SUBAPPLICATION GreenWhiteBackground_Seitenschieber (* Subapplication Type *)
  (* Standard: 61499-2 *)
  (* Version 1.0, 2023-02-06, franz *)
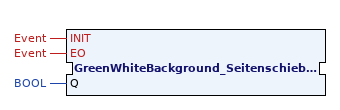
  EVENT_INPUT
    INIT;
    EO;
  END_EVENT
  VAR_INPUT
    Q : BOOL;
  END_VAR
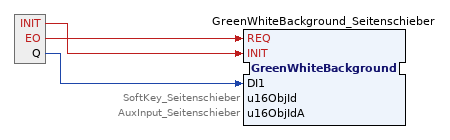
  SUBAPPS
    GreenWhiteBackground_Seitenschieber : GreenWhiteBackground(u16ObjId := SoftKey_Seitenschieber, u16ObjIdA := AuxInput_Seitenschieber);
  END_SUBAPPS
  EVENT_CONNECTIONS
    EO TO GreenWhiteBackground_Seitenschieber.REQ;
    INIT TO GreenWhiteBackground_Seitenschieber.INIT;
  END_CONNECTIONS
  DATA_CONNECTIONS
    Q TO GreenWhiteBackground_Seitenschieber.DI1;
  END_CONNECTIONS
END_SUBAPPLICATION
